SUBAPPLICATION Uebung_073 (* VDS auf UT ausgeben *)
  (* Standard: 61499-2; Description: Copyright (c) 2023 Meisterschulen am Ostbahnhof This program and the accompanying materials are made available under the terms of the Eclipse Public License 2.0 which is available at https://www.eclipse.org/legal/epl-2.0/ SPDX-License-Identifier: EPL-2.0 *)
  (* Version 1.0, 2023-10-23, Franz Höpfinger, Meisterschulen am Ostbahnhof *)
  IMPORT logiBUS::io::DI::logiBUS_DI;
  IMPORT logiBUS::io::DI::logiBUS_DI_Events;
  IMPORT logiBUS::io::DQ::logiBUS_DO;
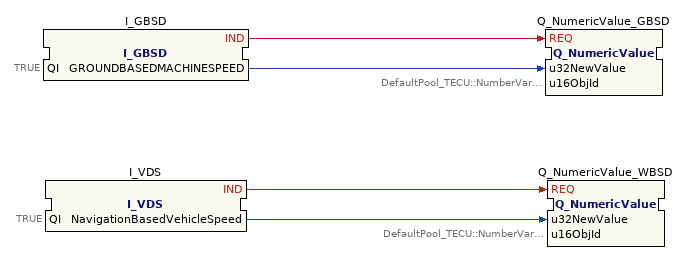
  FBS
    I_GBSD : isobus::tecu::I_GBSD(QI := TRUE);
    Q_NumericValue_GBSD : isobus::ut::Q_NumericValue(u16ObjId := DefaultPool_TECU::NumberVariable_Ground_based_machine_speed);
    I_VDS : isobus::tecu::I_VDS(QI := TRUE);
    Q_NumericValue_WBSD : isobus::ut::Q_NumericValue(u16ObjId := DefaultPool_TECU::NumberVariable_Wheel_based_machine_speed);
  END_FBS
  EVENT_CONNECTIONS
    I_GBSD.IND TO Q_NumericValue_GBSD.REQ;
    I_VDS.IND TO Q_NumericValue_WBSD.REQ;
  END_CONNECTIONS
  DATA_CONNECTIONS
    I_GBSD.GROUNDBASEDMACHINESPEED TO Q_NumericValue_GBSD.u32NewValue;
    I_VDS.NavigationBasedVehicleSpeed TO Q_NumericValue_WBSD.u32NewValue;
  END_CONNECTIONS
END_SUBAPPLICATION
